Universal Robots URScript: T011_qwen2.5-coder_32b_baseline_rep1.urscript

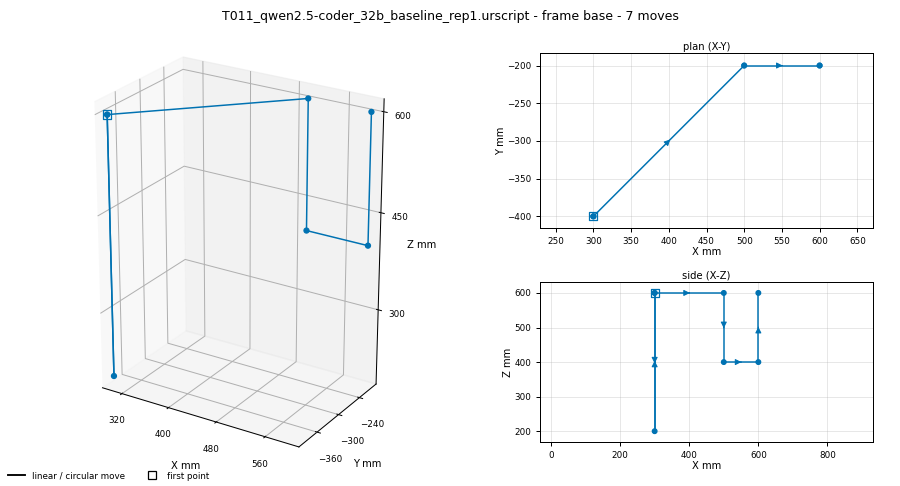
[picture p0: tool path of T011_qwen2.5-coder_32b_baseline_rep1.urscript in frame base, 7 of 8 moves have a stored position in this frame; points joined in program order, loops and branches not executed]
def dual_zone_pick_place():
    # Set payload and max speed
    set_payload(1.2, [0,0,0,0,0,0])
    set_tcp_speed_limit(300)

    # Move to Home position
    movej(get_inverse_kin([0.0, -pi/2, pi/2, 0.0, pi/2, 0.0]), a=1.4, v=1.05)

    # Move above storage bin
    movel(p[0.3, -0.4, 0.6, 3.14, 0, 0], a=1.2, v=0.28)

    # Descend to pick position
    movel(p[0.3, -0.4, 0.2, 3.14, 0, 0], a=1.2, v=0.12)

    # Lift from bin
    movel(p[0.3, -0.4, 0.6, 3.14, 0, 0], a=1.2, v=0.2)

    # Transit to handoff zone
    movel(p[0.5, -0.2, 0.6, 3.14, 0, 0], a=1.2, v=0.25)

    # Placeholder for next moves (3 more)
    # Move in handoff zone
    movel(p[0.5, -0.2, 0.4, 3.14, 0, 0], a=1.2, v=0.25)
    movel(p[0.6, -0.2, 0.4, 3.14, 0, 0], a=1.2, v=0.25)
    movel(p[0.6, -0.2, 0.6, 3.14, 0, 0], a=1.2, v=0.25)

end
